// TIA Portal V21 export
TYPE "Std_Sensore"
   STRUCT
      In : Struct
         Stato : Bool;
      END_STRUCT;
      Prm : Struct
         UnitàMisura : "Std_UnitàDiMisura";
      END_STRUCT;
      Hmi : Struct
         ForzaPos : Bool;
         ForzaNeg : Bool;
      END_STRUCT;
      Allarmi : Struct
         "A" : Array[0.."K_NumAllarmiPerSensori"] of "Std_PrmAllarmeStd";
         WordHMI : Word := 16#0000;
      END_STRUCT;
      Out : Struct
         PresProd : Bool;
         Allarmi : Struct
            "A" : Array[0.."K_NumAllarmiPerMotori"] of "Std_PrmAllarmeStd";
            WordHMI : Word := 16#0000;
         END_STRUCT;
      END_STRUCT;
      Rif_Inc : Struct
         K_Zona : Int;
      END_STRUCT;
   END_STRUCT;
END_TYPE
